// TIA Portal project "Warehouse Automated" (V17)

(* hardware
DEVICE "S7-300/ET200M station_1"  S7-300 station
   slot 0: "Rail_0"  Rail  6ES7 390-1***0-0AA0
   slot 2: "PLC_1"  CPU 313C-2 DP  6ES7 313-6CG04-0AB0  V3.3
      slot 0: "MPI interface_1"  MPI
      slot 1: "DP interface_1"  DP
      slot 2: "DI 16/DO 16_1"  DI16/DO16
      slot 4: "Count_1"  Counter
*)

// ===== PLC "PLC_1"  CPU 313C-2 DP =====

VAR_GLOBAL   // PLC tag table "Tag table_1"
   "At Entry" AT %I0.0 : Bool;
   "At Load" AT %I0.1 : Bool;
   "At Left" AT %I0.2 : Bool;
   "At Middle" AT %I0.3 : Bool;
   "At Right" AT %I0.4 : Bool;
   "At Unload" AT %I0.5 : Bool;
   "At Exit" AT %I0.6 : Bool;
   "Moving X" AT %I0.7 : Bool;
   "Moving Z" AT %I1.0 : Bool;
   "Start" AT %I1.1 : Bool;
   "Reset" AT %I1.2 : Bool;
   "Stop" AT %I1.3 : Bool;
   "Emergency stop" AT %I1.4 : Bool;
   "Auto" AT %I1.5 : Bool;
   "Entry Conveyor" AT %Q0.0 : Bool;
   "Load Conveyor" AT %Q0.1 : Bool;
   "Forks Left" AT %Q0.2 : Bool;
   "Forks Right" AT %Q0.3 : Bool;
   "Lift" AT %Q0.4 : Bool;
   "Unload Conveyor" AT %Q0.5 : Bool;
   "Exit Conveyor" AT %Q0.6 : Bool;
   "Start Light" AT %Q0.7 : Bool;
   "Reset Light" AT %Q1.0 : Bool;
   "Stop Light" AT %Q1.1 : Bool;
   "target position" AT %QD30 : DInt;
   "State 1" AT %M0.1 : Bool;
   "State 2" AT %M0.2 : Bool;
   "State 3" AT %M0.3 : Bool;
   "State 4" AT %M0.4 : Bool;
   "State 5" AT %M0.5 : Bool;
   "State 6" AT %M0.6 : Bool;
   "State 7" AT %M0.7 : Bool;
   "State 8" AT %M1.0 : Bool;
   "State 9" AT %M1.1 : Bool;
   "t" AT %MD30 : DWord;
   "State 0" AT %M0.0 : Bool;
END_VAR

VAR_GLOBAL   // PLC tag table "Default tag table"
   "a0" AT %M1.2 : Bool;
   "a1" AT %M1.3 : Bool;
   "a2" AT %M1.4 : Bool;
   "a3" AT %M1.5 : Bool;
   "a4" AT %M1.6 : Bool;
   "a5" AT %M1.7 : Bool;
END_VAR

FUNCTION "Start Stop" : Void   // FC1, LAD
{ S7_Optimized_Access := 'FALSE' }
VERSION : 0.1
BEGIN

REGION Network 1
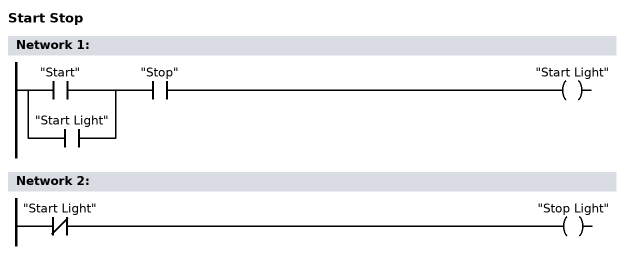
   RUNG wire#powerrail
      Contact( "Start" )
      wire#w1
      Contact( "Stop" )
      Coil( "Start Light" )
   END_RUNG
   RUNG wire#powerrail
      Contact( "Start Light" )
   END_RUNG wire#w1
   // the same network as SCL:
   "Start Light" := ("Start" OR "Start Light") AND "Stop";
END_REGION

REGION Network 2
   RUNG wire#powerrail
      I_Contact( "Start Light" )
      Coil( "Stop Light" )
   END_RUNG
   // the same network as SCL:
   "Stop Light" := NOT "Start Light";
END_REGION
END_FUNCTION

FUNCTION "States" : Void   // FC2, LAD
{ S7_Optimized_Access := 'FALSE' }
VERSION : 0.1
   VAR_TEMP   // added for the SCL form of the ladder/FBD networks
      _w1 : Bool;
      _w2 : Bool;
   END_VAR
BEGIN

REGION Network 1
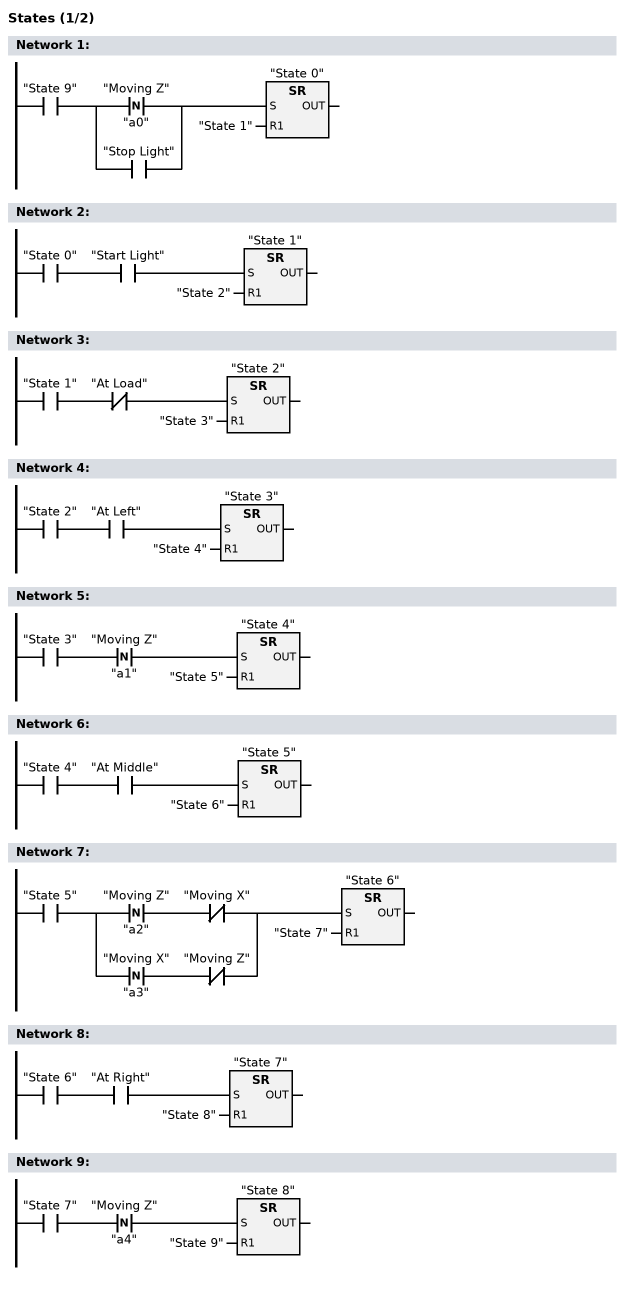
   RUNG wire#powerrail
      Contact( "State 9" )
      wire#w1
      N_Contact(operand := "Moving Z", bit := "a0")
      wire#w2
      S_SR(operand := "State 0", r1 := "State 1")
   END_RUNG
   RUNG wire#w1
      Contact( "Stop Light" )
   END_RUNG wire#w2
   // the same network as SCL:
   #_w1 := "State 9" AND NOT "Moving Z" AND "a0";   // falling edge of "Moving Z"
   "a0" := "Moving Z";
   IF #_w1 OR ("State 9" AND "Stop Light") THEN
       "State 0" := TRUE;   // SR flip-flop
   END_IF;
   IF "State 1" THEN "State 0" := FALSE; END_IF;
END_REGION

REGION Network 2
   RUNG wire#powerrail
      Contact( "State 0" )
      Contact( "Start Light" )
      S_SR(operand := "State 1", r1 := "State 2")
   END_RUNG
   // the same network as SCL:
   IF "State 0" AND "Start Light" THEN
       "State 1" := TRUE;   // SR flip-flop
   END_IF;
   IF "State 2" THEN "State 1" := FALSE; END_IF;
END_REGION

REGION Network 3
   RUNG wire#powerrail
      Contact( "State 1" )
      I_Contact( "At Load" )
      S_SR(operand := "State 2", r1 := "State 3")
   END_RUNG
   // the same network as SCL:
   IF "State 1" AND NOT "At Load" THEN
       "State 2" := TRUE;   // SR flip-flop
   END_IF;
   IF "State 3" THEN "State 2" := FALSE; END_IF;
END_REGION

REGION Network 4
   RUNG wire#powerrail
      Contact( "State 2" )
      Contact( "At Left" )
      S_SR(operand := "State 3", r1 := "State 4")
   END_RUNG
   // the same network as SCL:
   IF "State 2" AND "At Left" THEN
       "State 3" := TRUE;   // SR flip-flop
   END_IF;
   IF "State 4" THEN "State 3" := FALSE; END_IF;
END_REGION

REGION Network 5
   RUNG wire#powerrail
      Contact( "State 3" )
      N_Contact(operand := "Moving Z", bit := "a1")
      S_SR(operand := "State 4", r1 := "State 5")
   END_RUNG
   // the same network as SCL:
   #_w1 := "State 3" AND NOT "Moving Z" AND "a1";   // falling edge of "Moving Z"
   "a1" := "Moving Z";
   IF #_w1 THEN
       "State 4" := TRUE;   // SR flip-flop
   END_IF;
   IF "State 5" THEN "State 4" := FALSE; END_IF;
END_REGION

REGION Network 6
   RUNG wire#powerrail
      Contact( "State 4" )
      Contact( "At Middle" )
      S_SR(operand := "State 5", r1 := "State 6")
   END_RUNG
   // the same network as SCL:
   IF "State 4" AND "At Middle" THEN
       "State 5" := TRUE;   // SR flip-flop
   END_IF;
   IF "State 6" THEN "State 5" := FALSE; END_IF;
END_REGION

REGION Network 7
   RUNG wire#powerrail
      Contact( "State 5" )
      wire#w1
      N_Contact(operand := "Moving Z", bit := "a2")
      I_Contact( "Moving X" )
      wire#w2
      S_SR(operand := "State 6", r1 := "State 7")
   END_RUNG
   RUNG wire#w1
      N_Contact(operand := "Moving X", bit := "a3")
      I_Contact( "Moving Z" )
   END_RUNG wire#w2
   // the same network as SCL:
   #_w1 := "State 5" AND NOT "Moving Z" AND "a2";   // falling edge of "Moving Z"
   "a2" := "Moving Z";
   #_w2 := "State 5" AND NOT "Moving X" AND "a3";   // falling edge of "Moving X"
   "a3" := "Moving X";
   IF (#_w1 AND NOT "Moving X") OR (#_w2 AND NOT "Moving Z") THEN
       "State 6" := TRUE;   // SR flip-flop
   END_IF;
   IF "State 7" THEN "State 6" := FALSE; END_IF;
END_REGION

REGION Network 8
   RUNG wire#powerrail
      Contact( "State 6" )
      Contact( "At Right" )
      S_SR(operand := "State 7", r1 := "State 8")
   END_RUNG
   // the same network as SCL:
   IF "State 6" AND "At Right" THEN
       "State 7" := TRUE;   // SR flip-flop
   END_IF;
   IF "State 8" THEN "State 7" := FALSE; END_IF;
END_REGION

REGION Network 9
   RUNG wire#powerrail
      Contact( "State 7" )
      N_Contact(operand := "Moving Z", bit := "a4")
      S_SR(operand := "State 8", r1 := "State 9")
   END_RUNG
   // the same network as SCL:
   #_w1 := "State 7" AND NOT "Moving Z" AND "a4";   // falling edge of "Moving Z"
   "a4" := "Moving Z";
   IF #_w1 THEN
       "State 8" := TRUE;   // SR flip-flop
   END_IF;
   IF "State 9" THEN "State 8" := FALSE; END_IF;
END_REGION

REGION Network 10
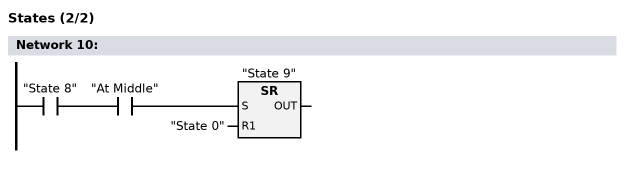
   RUNG wire#powerrail
      Contact( "State 8" )
      Contact( "At Middle" )
      S_SR(operand := "State 9", r1 := "State 0")
   END_RUNG
   // the same network as SCL:
   IF "State 8" AND "At Middle" THEN
       "State 9" := TRUE;   // SR flip-flop
   END_IF;
   IF "State 0" THEN "State 9" := FALSE; END_IF;
END_REGION
END_FUNCTION

FUNCTION "Actuators" : Void   // FC3, LAD
{ S7_Optimized_Access := 'FALSE' }
VERSION : 0.1
   VAR_TEMP   // added for the SCL form of the ladder/FBD networks
      _w1 : Bool;
   END_VAR
BEGIN

REGION Network 1
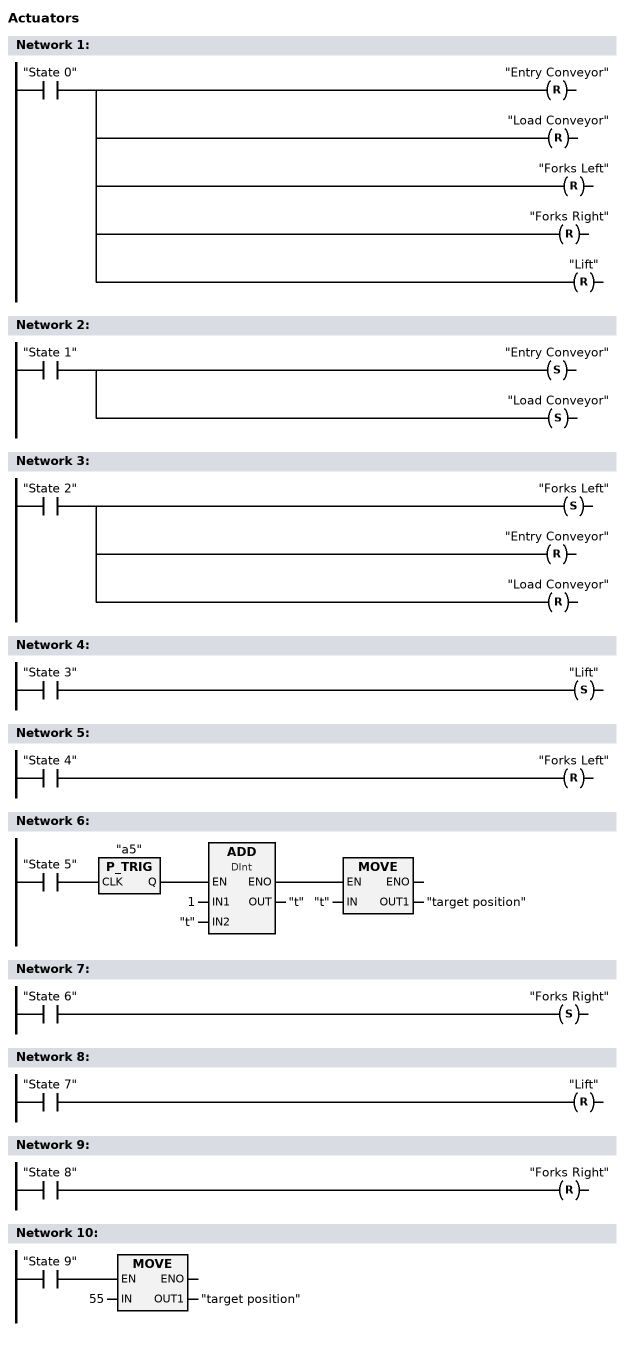
   RUNG wire#powerrail
      Contact( "State 0" )
      wire#w1
      R_Coil( "Entry Conveyor" )
   END_RUNG
   RUNG wire#w1
      R_Coil( "Load Conveyor" )
   END_RUNG
   RUNG wire#w1
      R_Coil( "Forks Left" )
   END_RUNG
   RUNG wire#w1
      R_Coil( "Forks Right" )
   END_RUNG
   RUNG wire#w1
      R_Coil( "Lift" )
   END_RUNG
   // the same network as SCL:
   IF "State 0" THEN
       "Entry Conveyor" := FALSE;
       "Load Conveyor" := FALSE;
       "Forks Left" := FALSE;
       "Forks Right" := FALSE;
       "Lift" := FALSE;
   END_IF;
END_REGION

REGION Network 2
   RUNG wire#powerrail
      Contact( "State 1" )
      wire#w1
      S_Coil( "Entry Conveyor" )
   END_RUNG
   RUNG wire#w1
      S_Coil( "Load Conveyor" )
   END_RUNG
   // the same network as SCL:
   IF "State 1" THEN
       "Entry Conveyor" := TRUE;
       "Load Conveyor" := TRUE;
   END_IF;
END_REGION

REGION Network 3
   RUNG wire#powerrail
      Contact( "State 2" )
      wire#w1
      S_Coil( "Forks Left" )
   END_RUNG
   RUNG wire#w1
      R_Coil( "Entry Conveyor" )
   END_RUNG
   RUNG wire#w1
      R_Coil( "Load Conveyor" )
   END_RUNG
   // the same network as SCL:
   IF "State 2" THEN
       "Forks Left" := TRUE;
       "Entry Conveyor" := FALSE;
       "Load Conveyor" := FALSE;
   END_IF;
END_REGION

REGION Network 4
   RUNG wire#powerrail
      Contact( "State 3" )
      S_Coil( "Lift" )
   END_RUNG
   // the same network as SCL:
   IF "State 3" THEN "Lift" := TRUE; END_IF;
END_REGION

REGION Network 5
   RUNG wire#powerrail
      Contact( "State 4" )
      R_Coil( "Forks Left" )
   END_RUNG
   // the same network as SCL:
   IF "State 4" THEN "Forks Left" := FALSE; END_IF;
END_REGION

REGION Network 6
   RUNG wire#powerrail
      Contact( "State 5" )
      P_Trig( "a5" )
      { S7_Templates := "SrcType := DInt"; S7_GenerateENO := "TRUE" } Add(in1 := 1, in2 := "t", out => "t")
      { S7_GenerateENO := "TRUE" } Move(in := "t", out1 => "target position")
   END_RUNG
   // the same network as SCL:
   // ENO of a box is taken as its EN; it also drops when the box reports an error
   #_w1 := "State 5" AND NOT "a5";   // rising edge
   "a5" := "State 5";
   IF #_w1 THEN
       "t" := 1 + "t";
       "target position" := "t";
   END_IF;
END_REGION

REGION Network 7
   RUNG wire#powerrail
      Contact( "State 6" )
      S_Coil( "Forks Right" )
   END_RUNG
   // the same network as SCL:
   IF "State 6" THEN "Forks Right" := TRUE; END_IF;
END_REGION

REGION Network 8
   RUNG wire#powerrail
      Contact( "State 7" )
      R_Coil( "Lift" )
   END_RUNG
   // the same network as SCL:
   IF "State 7" THEN "Lift" := FALSE; END_IF;
END_REGION

REGION Network 9
   RUNG wire#powerrail
      Contact( "State 8" )
      R_Coil( "Forks Right" )
   END_RUNG
   // the same network as SCL:
   IF "State 8" THEN "Forks Right" := FALSE; END_IF;
END_REGION

REGION Network 10
   RUNG wire#powerrail
      Contact( "State 9" )
      { S7_GenerateENO := "TRUE" } Move(in := 55, out1 => "target position")
   END_RUNG
   // the same network as SCL:
   IF "State 9" THEN "target position" := 55; END_IF;
END_REGION
END_FUNCTION

ORGANIZATION_BLOCK "Main"   // OB1, LAD
TITLE = "Main Program Sweep (Cycle)"
{ S7_Optimized_Access := 'FALSE' }
VERSION : 0.1
   VAR_TEMP
      OB1_EV_CLASS : Byte;   // Bits 0-3 = 1 (Coming event), Bits 4-7 = 1 (Event class 1)
      OB1_SCAN_1 : Byte;   // 1 (Cold restart scan 1 of OB 1), 3 (Scan 2-n of OB 1)
      OB1_PRIORITY : Byte;   // Priority of OB Execution
      OB1_OB_NUMBR : Byte;   // 1 (Organization block 1, OB1)
      OB1_RESERVED_1 : Byte;   // Reserved for system
      OB1_RESERVED_2 : Byte;   // Reserved for system
      OB1_PREV_CYCLE : Int;   // Cycle time of previous OB1 scan (milliseconds)
      OB1_MIN_CYCLE : Int;   // Minimum cycle time of OB1 (milliseconds)
      OB1_MAX_CYCLE : Int;   // Maximum cycle time of OB1 (milliseconds)
      OB1_DATE_TIME : Date_And_Time;   // Date and time OB1 started
   END_VAR
BEGIN

REGION Network 1
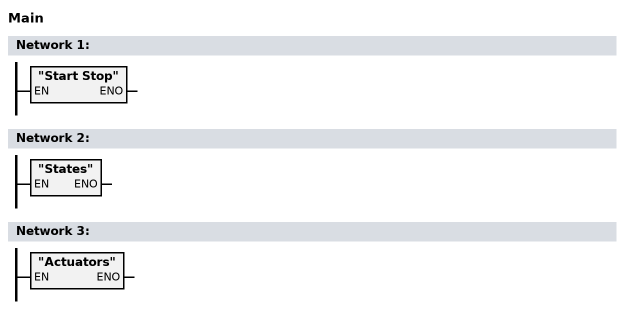
   RUNG wire#powerrail
      "Start Stop"()
   END_RUNG
   // the same network as SCL:
   "Start Stop"();
END_REGION

REGION Network 2
   RUNG wire#powerrail
      "States"()
   END_RUNG
   // the same network as SCL:
   "States"();
END_REGION

REGION Network 3
   RUNG wire#powerrail
      "Actuators"()
   END_RUNG
   // the same network as SCL:
   "Actuators"();
END_REGION
END_ORGANIZATION_BLOCK

ORGANIZATION_BLOCK "COMPLETE RESTART"   // OB100, LAD
TITLE = "Complete Restart"
{ S7_Optimized_Access := 'FALSE' }
VERSION : 0.1
   VAR_TEMP
      OB100_EV_CLASS : Byte;   // 16#13, Event class 1, Entering event state, Event logged in diagnostic buffer
      OB100_STRTUP : Byte;   // 16#81/82/83/84 Method of startup
      OB100_PRIORITY : Byte;   // Priority of OB Execution
      OB100_OB_NUMBR : Byte;   // 100 (Organization block 100, OB100)
      OB100_RESERVED_1 : Byte;   // Reserved for system
      OB100_RESERVED_2 : Byte;   // Reserved for system
      OB100_STOP : Word;   // Event that caused CPU to stop (16#4xxx)
      OB100_STRT_INFO : DWord;   // Information on how system started
      OB100_DATE_TIME : Date_And_Time;   // Date and time OB100 started
   END_VAR
BEGIN

REGION Network 1
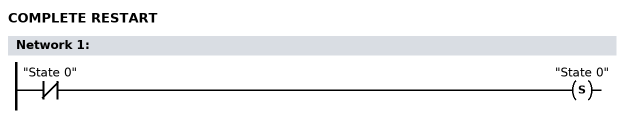
   RUNG wire#powerrail
      I_Contact( "State 0" )
      S_Coil( "State 0" )
   END_RUNG
   // the same network as SCL:
   IF NOT "State 0" THEN "State 0" := TRUE; END_IF;
END_REGION
END_ORGANIZATION_BLOCK